FUNCTION CallThisSingleTimeEachCycle : BOOL


TaskHeartbeat(update := TRUE);

END_FUNCTION

(* stored: Version 1.1.0.1, ProductVersion 3.1.4024.12
   POU CallThisSingleTimeEachCycle: Id {17bc738b-5835-46a1-928e-ac82fd18c60a}, SpecialFunc None *)
